// TwinCAT 3 PLC project Inspection_Control
// ProgramVersion: 3.1.4026.20
// libraries:
//   Core, * (Beckhoff Automation LLC)
//   CoreVision, * (Beckhoff Automation LLC)
//   Tc2_Standard, * (Beckhoff Automation GmbH)
//   Tc2_System, * (Beckhoff Automation GmbH)
//   Tc3_PackML_V3, * (Beckhoff Automation GmbH)
//   Nestle Vanguard Base Library, * (Nestle)
// project tree:
//   GVLs/ GVL_Vision.TcGVL
//   Module/ Vision_Inspection_HMI.TcPOU, Vision_Inspection_Module.TcPOU
//   / PlcTask.TcTTO (not stored), VisionTask.TcTTO (not stored)
//   POUs/ MAIN.TcPOU, Vision.TcPOU (not stored)
//   States/ ExecuteProduction.TcPOU, ExecuteManual.TcPOU, Starting.TcPOU, Stopping.TcPOU

// ---- GVLs/GVL_Vision.TcGVL
{attribute 'qualified_only'}
VAR_GLOBAL
	waferInspectionRecipe : WaferInspection;
	Camera : SimpleCamera;
	WaferDetectionProcess : ProcessSKU;
	ImageChannel : VisionChannel(Name := 'Beckhoff Camera', ImageSource := Camera, ImageProcess := WaferDetectionProcess);
END_VAR

// ---- Module/Vision_Inspection_HMI.TcPOU
FUNCTION_BLOCK Vision_Inspection_HMI EXTENDS StateControllerHMI
VAR
END_VAR

PROPERTY ControlObject : I_Base
SET
END_SET
END_PROPERTY

METHOD CyclicLogic
VAR_INST
	StartRT : R_TRIG;
	StopRT	: R_TRIG;
	ResetRT : R_TRIG;
END_VAR
SUPER^.CyclicLogic();

// User buttons
Statemachine_HMI.StartPermissive := Statemachine_HMI.CurrentState = E_PMLState.Idle;
Statemachine_HMI.StopPermissive	 := Statemachine_HMI.CurrentState <> E_PMLState.Aborted;
Statemachine_HMI.ResetPermissive := Statemachine_HMI.CurrentState = E_PMLState.Aborted OR Statemachine_HMI.CurrentState = E_PMLState.Stopped;
StartRT(CLK := Statemachine_HMI.StartPressed);
IF StartRT.Q THEN
	_stateMachine.RequestStart();
END_IF

StopRT(CLK := Statemachine_HMI.StopPressed);
IF StopRT.Q THEN
	IF Statemachine_HMI.CurrentState = E_PMLState.Stopped THEN
		_stateMachine.RequestAbort();
	ELSE
		_stateMachine.RequestStop();
	END_IF
END_IF

ResetRT(CLK := Statemachine_HMI.ResetPressed);
IF ResetRT.Q THEN
	IF Statemachine_HMI.CurrentState = E_PMLState.Aborted THEN
		_stateMachine.RequestClear();
	ELSE
		_stateMachine.RequestReset();
	END_IF
END_IF
END_METHOD

END_FUNCTION_BLOCK

// ---- Module/Vision_Inspection_Module.TcPOU
FUNCTION_BLOCK Vision_Inspection_Module EXTENDS Module
VAR
	PackMLModeController : ModeController(StateController := PackMLStateMachine, 
											Production := Production, 
											Manual := Manual, 
											Maintainence := Maintainence);
	PackMLStateMachine : StateController(ModeController := PackMLModeController);
	HMI : Vision_Inspection_HMI('Vision Inspection',PackMLStateMachine,PackMLModeController);
	
	// states 
	ProductionExecute : ExecuteProduction(PackMLStateMachine);
	ProductionStarting : Starting;
	ProductionStopping : Stopping;
	ManualExecute : ExecuteManual(PackMLStateMachine);
	ManualStarting : Starting;
	ManualStopping : Stopping;
	
	Production : ProductionMode(Name := 'Mounting Production', StateMachine := PackMLStateMachine) := (Execute := ProductionExecute,
																										Starting := ProductionStarting,
																										Stopping := ProductionStopping);
	Manual : ManualMode(Name := 'Mounting Manual', StateMachine := PackMLStateMachine) := (Execute := ManualExecute,
																										Starting := ManualStarting,
																										Stopping := ManualStopping);
	Maintainence : MaintainenceMode(Name := 'Mounting Maintainence', StateMachine := PackMLStateMachine);
	
	ChannelControl : VisionChannelControl(Name := 'Beckhoff Camera Control',VisionChannel := GVL_Vision.ImageChannel);
	
END_VAR

(* This Module will be done initialize when ModuleInitialized := TRUE;, subequently all subitems will be called to be initialized *)
METHOD Initializing
CyclicRunner.AddCallee(PackMLModeController);
CyclicRunner.AddCallee(PackMLStateMachine);
CyclicRunner.AddCallee(HMI);
CyclicRunner.AddCallee(ChannelControl);

ProductionExecute.SetDependencies(Control := ChannelControl);
ProductionStarting.SetDependencies(Control := ChannelControl);
ProductionStopping.SetDependencies(Control := ChannelControl);
END_METHOD

METHOD OnCyclicCall
END_METHOD

END_FUNCTION_BLOCK

// ---- States/ExecuteProduction.TcPOU
FUNCTION_BLOCK ExecuteProduction EXTENDS Vanguard_WaferDetection.State
VAR
	_stateMachine : I_ExecuteTranisitons;
	ChannelControl : I_VisionChannelControl;
	OperatingState : INT;
	SKUDetected : BOOL;
	startTrig : R_TRIG;
	stopTrig : R_TRIG;
	skuTrigger : R_TRIG;
END_VAR

METHOD Executing : BOOL
skuTrigger(CLK := SKUDetected);
CASE OperatingState OF 
	0:
		IF skuTrigger.Q THEN
			ChannelControl.TriggerImage();
			OperatingState := 1;
		END_IF
	1:
		IF ChannelControl.ImageProcessing THEN
			OperatingState := 2;
		END_IF
	2:
		IF ChannelControl.ImageProcessingCompletedSuccessfully THEN
			OperatingState := 0;
		ELSE
			OperatingState := 99;
		END_IF
END_CASE
END_METHOD

//FB_Init is always available implicitly and it is used primarily for initialization.
//The return value is not evaluated. For a specific influence, you can also declare the
//methods explicitly and provide additional code there with the standard initialization
//code. You can evaluate the return value.
METHOD FB_Init: BOOL
VAR_INPUT
    bInitRetains: BOOL; // TRUE: the retain variables are initialized (reset warm / reset cold)
    bInCopyCode: BOOL;  // TRUE: the instance will be copied to the copy code afterward (online change)   
	StateMachine : I_ExecuteTranisitons;
END_VAR
_stateMachine := StateMachine;
END_METHOD

METHOD SetDependencies : BOOL
VAR_INPUT
	Control : I_VisionChannelControl;
END_VAR
ChannelControl := Control;
END_METHOD

END_FUNCTION_BLOCK

// ---- States/Starting.TcPOU
FUNCTION_BLOCK Starting EXTENDS Vanguard_WaferDetection.State
VAR
	StartupState : INT;
	ChannelControl : I_VisionChannelControl;
END_VAR

METHOD Executing : BOOL
CASE StartupState OF
// 	0: //Unknown conditions
// 		IF SUCCEEDED(GVL_Vision.LabelProcess.LoadRecipe(WaferDetectRecipe)) THEN
// 			SystemReady := TRUE;
// 			StartupState := 1;
// 		END_IF

	0:
		IF ChannelControl.StartVision() THEN
			StartupState := 1;
		END_IF
	1:
		StartupState := 0;
		Executing := TRUE;
END_CASE
END_METHOD

METHOD SetDependencies : BOOL
VAR_INPUT
	Control : I_VisionChannelControl;
END_VAR
ChannelControl := Control;
END_METHOD

END_FUNCTION_BLOCK

// ---- States/Stopping.TcPOU
FUNCTION_BLOCK Stopping EXTENDS Vanguard_WaferDetection.State
VAR
	ShutdownState : INT;
	ChannelControl : I_VisionChannelControl;
END_VAR

METHOD Executing : BOOL
CASE ShutdownState OF		
	0: //unkown conditions
		IF ChannelControl.StopVision() THEN
			ShutdownState := 1;
		END_IF
	1:
		Executing := TRUE;
		ShutdownState := 0;
END_CASE
END_METHOD

METHOD SetDependencies : BOOL
VAR_INPUT
	Control : I_VisionChannelControl;
END_VAR
ChannelControl := Control;
END_METHOD

END_FUNCTION_BLOCK

// ---- States/ExecuteManual.TcPOU
FUNCTION_BLOCK ExecuteManual EXTENDS Vanguard_WaferDetection.State
VAR
	_stateMachine : I_ExecuteTranisitons;
	ChannelControl : I_VisionChannelControl;
	OperatingState : INT;
	DummySKUDetectedSignal : BOOL;
	startTrig : R_TRIG;
	stopTrig : R_TRIG;
	skuTrigger : R_TRIG;
END_VAR

METHOD Executing : BOOL
skuTrigger(CLK := DummySKUDetectedSignal);
CASE OperatingState OF 
	0:
		IF skuTrigger.Q THEN
			ChannelControl.TriggerImage();
			OperatingState := 1;
		END_IF
	1:
		IF ChannelControl.ImageProcessing THEN
			OperatingState := 2;
		END_IF
	2:
		IF ChannelControl.ImageProcessingCompletedSuccessfully THEN
			OperatingState := 0;
		ELSE
			OperatingState := 99;
		END_IF
END_CASE
END_METHOD

//FB_Init is always available implicitly and it is used primarily for initialization.
//The return value is not evaluated. For a specific influence, you can also declare the
//methods explicitly and provide additional code there with the standard initialization
//code. You can evaluate the return value.
METHOD FB_Init: BOOL
VAR_INPUT
    bInitRetains: BOOL; // TRUE: the retain variables are initialized (reset warm / reset cold)
    bInCopyCode: BOOL;  // TRUE: the instance will be copied to the copy code afterward (online change)   
	StateMachine : I_ExecuteTranisitons;
END_VAR
_stateMachine := StateMachine;
END_METHOD

METHOD SetDependencies : BOOL
VAR_INPUT
	Control : I_VisionChannelControl;
END_VAR
ChannelControl := Control;
END_METHOD

END_FUNCTION_BLOCK

// ---- POUs/MAIN.TcPOU
PROGRAM MAIN
VAR
	WaferVisionModule : Vision_Inspection_Module(Name := 'Wafer Detection Module');
	Init : BOOL;
END_VAR

IF NOT Init THEN
	Init := TRUE;
	WaferVisionModule.Initialize();
	GVL_Vision.waferInspectionRecipe.VisionProcess.MedianFilterSize := 5;
	GVL_Vision.WaferDetectionProcess.LoadRecipe(Recipe := GVL_Vision.waferInspectionRecipe);
	RETURN;
END_IF

WaferVisionModule.CyclicLogic();

END_PROGRAM
